FUNCTION_BLOCK FB_LimitSwitchState
VAR_INPUT
	diInputs	:	DINT;
END_VAR
VAR_OUTPUT
	xHiLS	:	BOOL;
	xLoLS	:	BOOL;
	STO: BOOL;
END_VAR
VAR
	di_1: BOOL;
	di_2: BOOL;
	FLS: BOOL; //TRUE is active (ie. limit switch is hit, drive is configured normally-closed). This is bad.
	RLS: BOOL; 
	
END_VAR
VAR CONSTANT
	cHighVal	:	UDINT := 16#00010002;
	cLowVal		:	UDINT := 16#00020001;
END_VAR

(* ElmoMC Limit State
A. Wallace 2017-2-25

Sets the high and low limit switch bools based on input status dint from ElmoMC Drives *)


RLS		:= diInputs.0;
FLS		:= diInputs.1;

STO 	:= diInputs.3;

di_1	:= diInputs.16;
di_2	:= diInputs.17;

//

xHiLS := NOT FLS AND STO;
xLoLS := NOT RLS AND STO;

END_FUNCTION_BLOCK

(* stored: Version 1.1.0.1, ProductVersion 3.1.4020.12
   POU FB_LimitSwitchState: Id {b186eb7c-ca72-42e0-b2ec-6cc7d83a7a1f}, SpecialFunc None *)
